PROGRAM Axis03_Y_1
VAR
	Axis03: AXIS_REF;											//회전축
	Axis03_MC_Home: FB_HomeBeforeMoveAX8000;
	Axis03_MC_Power: MC_Power;
	Axis03_Status: MC_ReadStatus;
	Axis03_Position_Read: MC_ReadActualPosition;
	Axis03_Velocity_Read: MC_ReadActualVelocity;
	Axis03_Reset: MC_Reset;										//모터 알람 리셋
	Axis03_Stop: MC_Stop;										//모터 정지
	Axis03_Press_Move: MC_MoveAbsolute;
	Axis03_Home_Pos_Move: MC_MoveAbsolute;
	Axis03_Wait_Pos_Move: MC_MoveAbsolute;
	Axis03_Target_Pos_Move: MC_MoveAbsolute;
	Axis03_Work_End_Move: MC_MoveAbsolute;
	Axis03_Jog: MC_Jog;	
	
	
	Always_ON	:	BOOL	:=TRUE	;//상시 ON
	Always_OFF	:	BOOL	:=FALSE	;//상시 OFF
	Home_Interlock			:	BOOL	;
	Home_Pos_Interlock		: 	BOOL	;
	Wait_Pos_Interlock		:	BOOL	;
	Target_Pos_Interlock	:	BOOL	;
	Work_End_POs_Interlock	:	BOOL	;

	Axis03_Calibration: MC_MoveAbsolute;
	Axis03_Tool_Change: MC_MoveAbsolute;
END_VAR
VAR // added by the converter: edge detectors and wires of the graphical bodies
    _rt1, _rt2, _rt3, _rt4, _rt5 : R_TRIG;
    _w1, _w2 : BOOL;
END_VAR

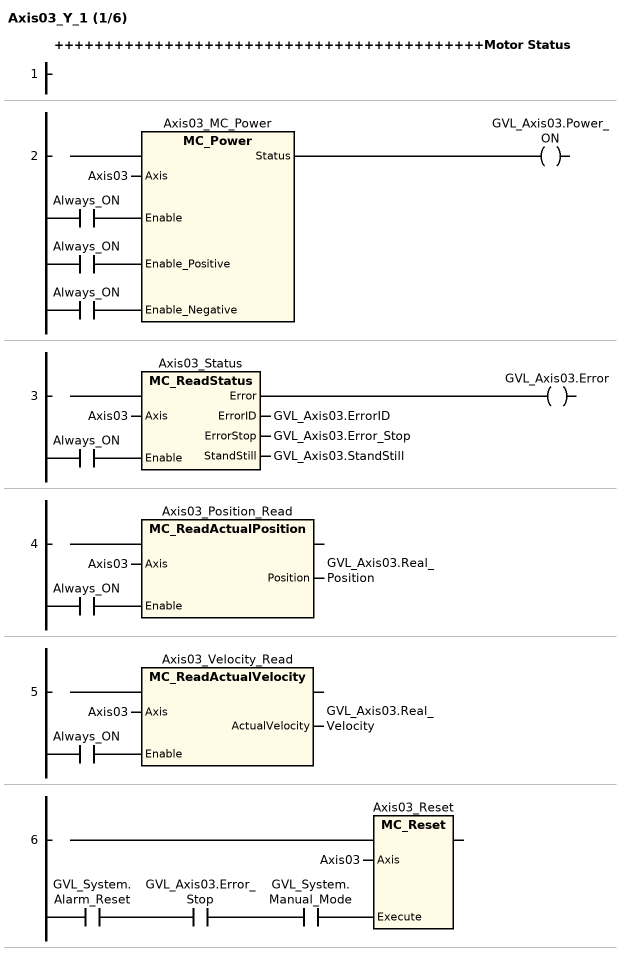
// NETWORK 1: +++++++++++++++++++++++++++++++++++++++++++Motor Status

// NETWORK 2
Axis03_MC_Power(
    Axis := Axis03,
    Enable := Always_ON,
    Enable_Positive := Always_ON,
    Enable_Negative := Always_ON); // MC_Power
GVL_Axis03.Power_ON := Axis03_MC_Power.Status;

// NETWORK 3
Axis03_Status(
    Axis := Axis03,
    Enable := Always_ON,
    Error => GVL_Axis03.Error,
    ErrorID => GVL_Axis03.ErrorID,
    ErrorStop => GVL_Axis03.Error_Stop,
    StandStill => GVL_Axis03.StandStill); // MC_ReadStatus

// NETWORK 4
Axis03_Position_Read(Axis := Axis03, Enable := Always_ON, Position => GVL_Axis03.Real_Position); // MC_ReadActualPosition

// NETWORK 5
Axis03_Velocity_Read(Axis := Axis03, Enable := Always_ON, ActualVelocity => GVL_Axis03.Real_Velocity); // MC_ReadActualVelocity

// NETWORK 6
Axis03_Reset(Axis := Axis03, Execute := GVL_System.Alarm_Reset AND GVL_Axis03.Error_Stop AND GVL_System.Manual_Mode); // MC_Reset

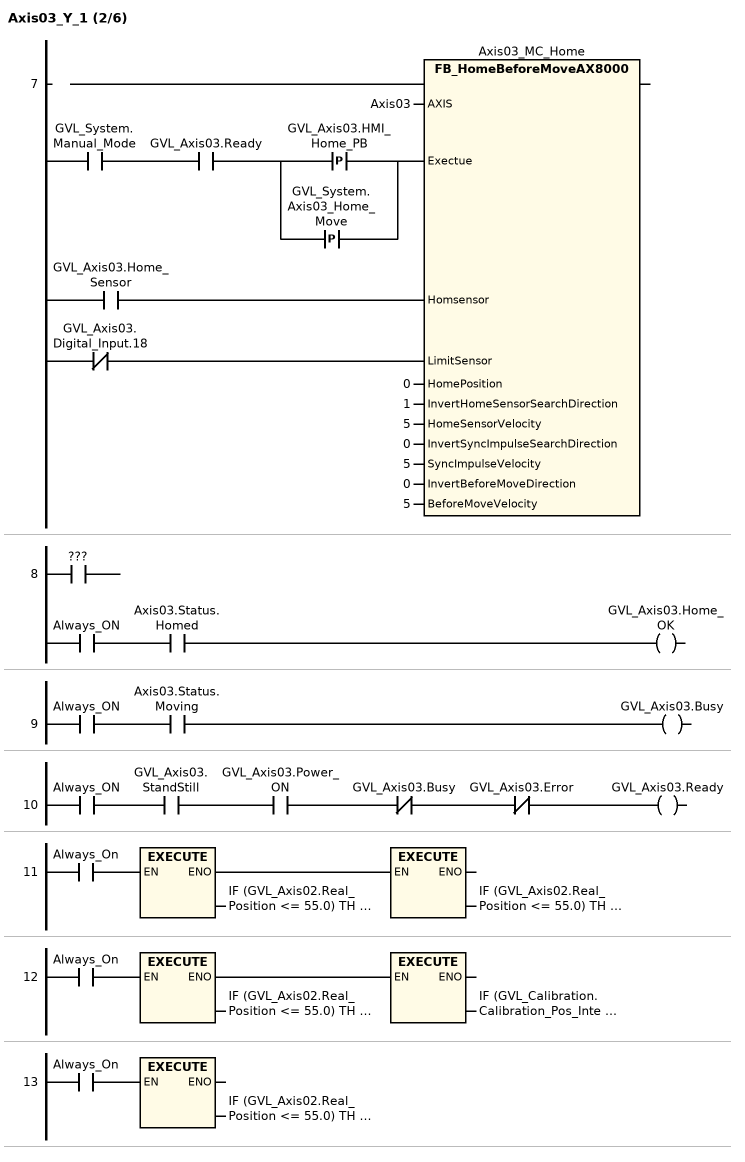
// NETWORK 7
_rt1(CLK := GVL_Axis03.HMI_Home_PB);
_rt2(CLK := GVL_System.Axis03_Home_Move);
Axis03_MC_Home(
    AXIS := Axis03,
    Exectue := GVL_System.Manual_Mode AND GVL_Axis03.Ready AND (_rt1.Q OR _rt2.Q),
    Homsensor := GVL_Axis03.Home_Sensor,
    LimitSensor := NOT GVL_Axis03.Digital_Input.18,
    HomePosition := 0,
    InvertHomeSensorSearchDirection := 1,
    HomeSensorVelocity := 5,
    InvertSyncImpulseSearchDirection := 0,
    SyncImpulseVelocity := 5,
    InvertBeforeMoveDirection := 0,
    BeforeMoveVelocity := 5); // FB_HomeBeforeMoveAX8000

// NETWORK 8
GVL_Axis03.Home_OK := Always_ON AND Axis03.Status.Homed;

// NETWORK 9
GVL_Axis03.Busy := Always_ON AND Axis03.Status.Moving;

// NETWORK 10
GVL_Axis03.Ready := Always_ON AND GVL_Axis03.StandStill AND GVL_Axis03.Power_ON AND NOT GVL_Axis03.Busy AND NOT GVL_Axis03.Error;

// NETWORK 11
_w1 := Always_On;
IF _w1 THEN
    IF (GVL_Axis02.Real_Position <= 55.0) THEN
        Home_Pos_Interlock := TRUE;
    ELSE
        IF (GVL_Axis03.Home_Position_Data >= 12.1) AND 
           (GVL_Axis03.Home_Position_Data <= 18.1) THEN
            Home_Pos_Interlock := TRUE;
        ELSE 
           Home_Pos_Interlock := FALSE;
        END_IF;
    END_IF;
END_IF
IF _w1 THEN
    IF (GVL_Axis02.Real_Position <= 55.0) THEN
        Wait_Pos_Interlock := TRUE;
    ELSE
        IF (GVL_Axis03.Wait_Position_Data >= 12.1) AND 
           (GVL_Axis03.Wait_Position_Data <= 18.1) THEN
            Wait_Pos_Interlock := TRUE;
        ELSE 
           Wait_Pos_Interlock := FALSE;
        END_IF;
    END_IF;
END_IF

// NETWORK 12
_w2 := Always_On;
IF _w2 THEN
    IF (GVL_Axis02.Real_Position <= 55.0) THEN
        Work_End_Pos_Interlock := TRUE;
    ELSE
        IF (GVL_Axis03.Work_End_Position_Data >= 12.1) AND 
           (GVL_Axis03.Work_End_Position_Data <= 18.1) THEN
            Work_End_Pos_Interlock := TRUE;
        ELSE 
           Work_End_Pos_Interlock := FALSE;
        END_IF;
    END_IF;
END_IF
IF _w2 THEN
    IF (GVL_Calibration.Calibration_Pos_Interlock = TRUE) AND (Home_Pos_Interlock = TRUE)
    AND (Wait_Pos_Interlock = TRUE) AND (Target_Pos_Interlock = TRUE) AND (Work_End_POs_Interlock = TRUE) THEN
    	GVL_Axis03.Interlock := TRUE;
    	ELSE
    	GVL_Axis03.Interlock := FALSE;	
    
    END_IF
END_IF

// NETWORK 13
IF Always_On THEN
    IF (GVL_Axis02.Real_Position <= 55.0) THEN
        Home_Interlock := TRUE;
    ELSE
        Home_Interlock := FALSE;
    
    END_IF;
END_IF

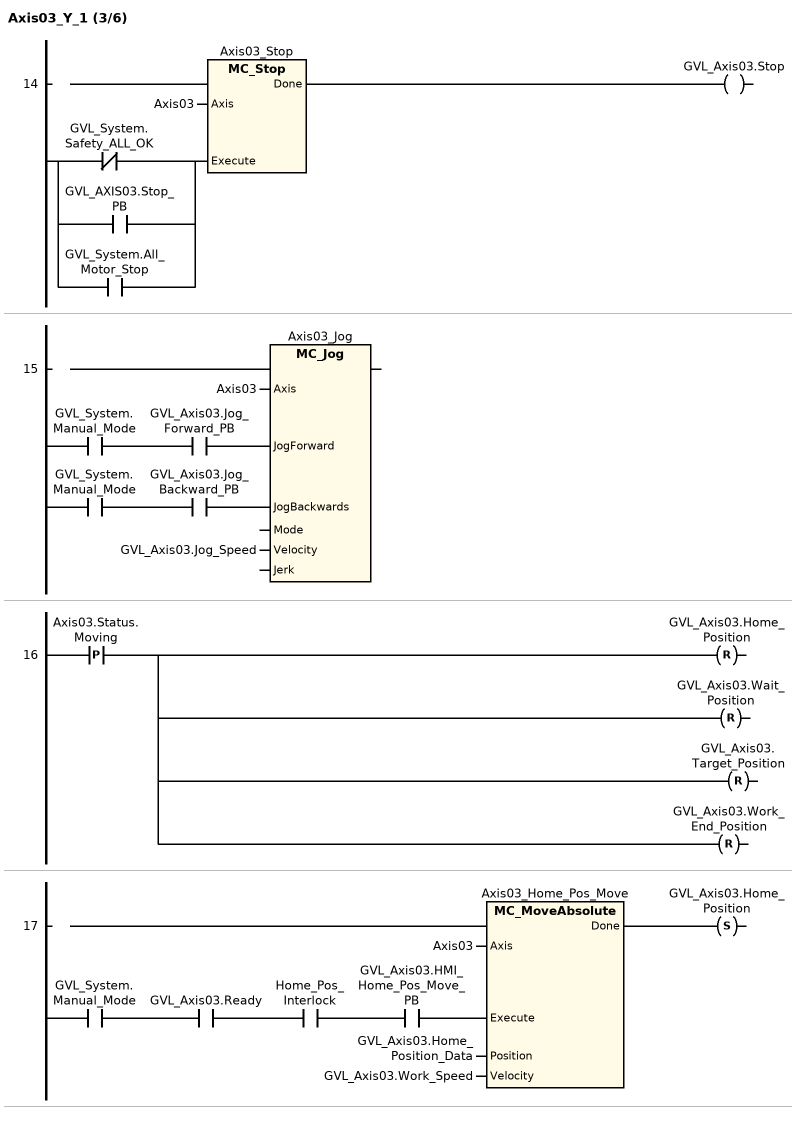
// NETWORK 14
Axis03_Stop(Axis := Axis03, Execute := NOT GVL_System.Safety_ALL_OK OR GVL_AXIS03.Stop_PB OR GVL_System.All_Motor_Stop); // MC_Stop
GVL_Axis03.Stop := Axis03_Stop.Done;

// NETWORK 15
Axis03_Jog(
    Axis := Axis03,
    JogForward := GVL_System.Manual_Mode AND GVL_Axis03.Jog_Forward_PB,
    JogBackwards := GVL_System.Manual_Mode AND GVL_Axis03.Jog_Backward_PB,
    Velocity := GVL_Axis03.Jog_Speed); // MC_Jog

// NETWORK 16
_rt3(CLK := Axis03.Status.Moving);
GVL_Axis03.Home_Position R= _rt3.Q;
GVL_Axis03.Wait_Position R= _rt3.Q;
GVL_Axis03.Target_Position R= _rt3.Q;
GVL_Axis03.Work_End_Position R= _rt3.Q;

// NETWORK 17
Axis03_Home_Pos_Move(
    Axis := Axis03,
    Execute := GVL_System.Manual_Mode AND GVL_Axis03.Ready AND Home_Pos_Interlock AND GVL_Axis03.HMI_Home_Pos_Move_PB,
    Position := GVL_Axis03.Home_Position_Data,
    Velocity := GVL_Axis03.Work_Speed); // MC_MoveAbsolute
GVL_Axis03.Home_Position S= Axis03_Home_Pos_Move.Done;

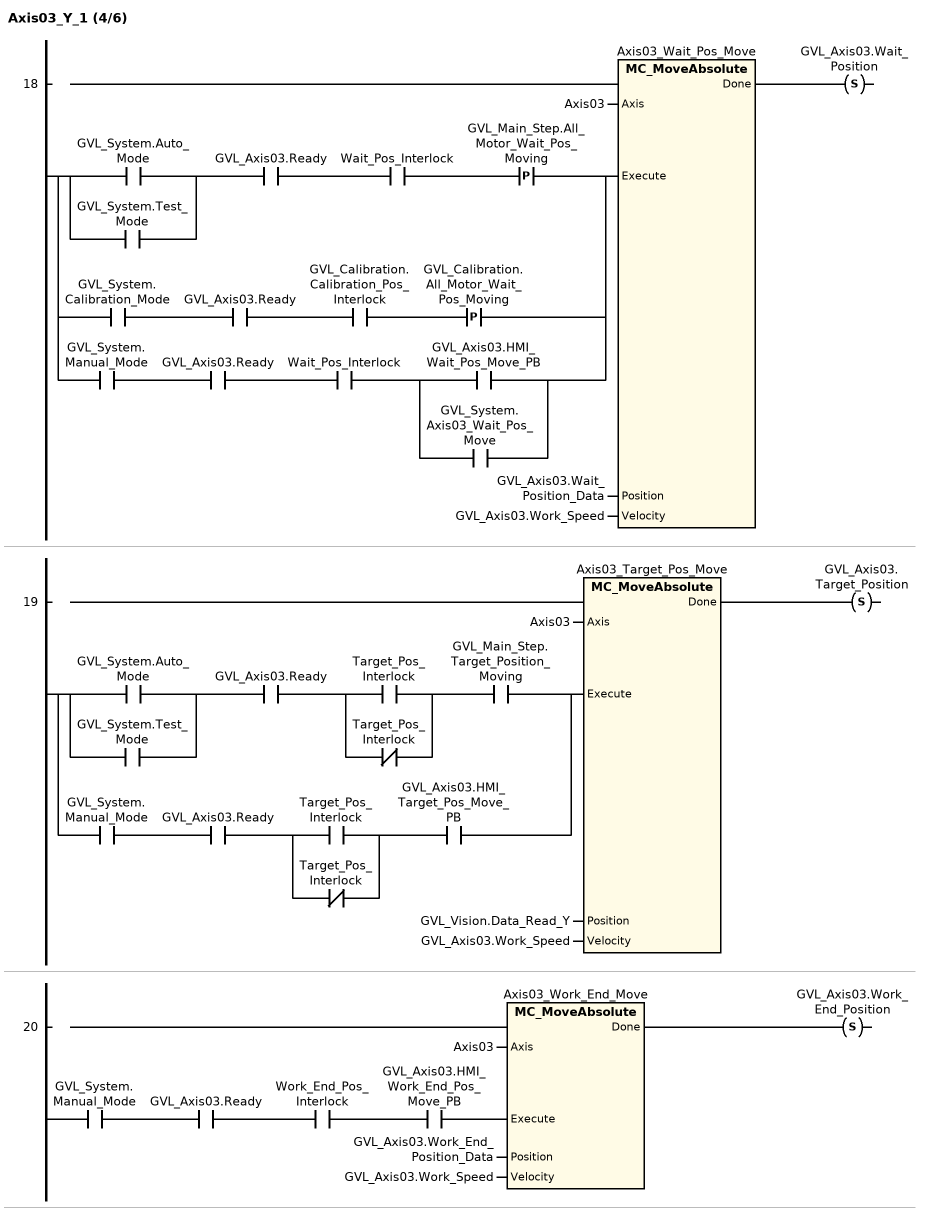
// NETWORK 18
_rt4(CLK := GVL_Main_Step.All_Motor_Wait_Pos_Moving);
_rt5(CLK := GVL_Calibration.All_Motor_Wait_Pos_Moving);
Axis03_Wait_Pos_Move(
    Axis := Axis03,
    Execute := (GVL_System.Auto_Mode OR GVL_System.Test_Mode) AND GVL_Axis03.Ready AND Wait_Pos_Interlock AND _rt4.Q OR GVL_System.Calibration_Mode AND GVL_Axis03.Ready AND GVL_Calibration.Calibration_Pos_Interlock AND _rt5.Q OR GVL_System.Manual_Mode AND GVL_Axis03.Ready AND Wait_Pos_Interlock AND (GVL_Axis03.HMI_Wait_Pos_Move_PB OR GVL_System.Axis03_Wait_Pos_Move),
    Position := GVL_Axis03.Wait_Position_Data,
    Velocity := GVL_Axis03.Work_Speed); // MC_MoveAbsolute
GVL_Axis03.Wait_Position S= Axis03_Wait_Pos_Move.Done;

// NETWORK 19
Axis03_Target_Pos_Move(
    Axis := Axis03,
    Execute := (GVL_System.Auto_Mode OR GVL_System.Test_Mode) AND GVL_Axis03.Ready AND (Target_Pos_Interlock OR NOT Target_Pos_Interlock) AND GVL_Main_Step.Target_Position_Moving OR GVL_System.Manual_Mode AND GVL_Axis03.Ready AND (Target_Pos_Interlock OR NOT Target_Pos_Interlock) AND GVL_Axis03.HMI_Target_Pos_Move_PB,
    Position := GVL_Vision.Data_Read_Y,
    Velocity := GVL_Axis03.Work_Speed); // MC_MoveAbsolute
GVL_Axis03.Target_Position S= Axis03_Target_Pos_Move.Done;

// NETWORK 20
Axis03_Work_End_Move(
    Axis := Axis03,
    Execute := GVL_System.Manual_Mode AND GVL_Axis03.Ready AND Work_End_Pos_Interlock AND GVL_Axis03.HMI_Work_End_Pos_Move_PB,
    Position := GVL_Axis03.Work_End_Position_Data,
    Velocity := GVL_Axis03.Work_Speed); // MC_MoveAbsolute
GVL_Axis03.Work_End_Position S= Axis03_Work_End_Move.Done;

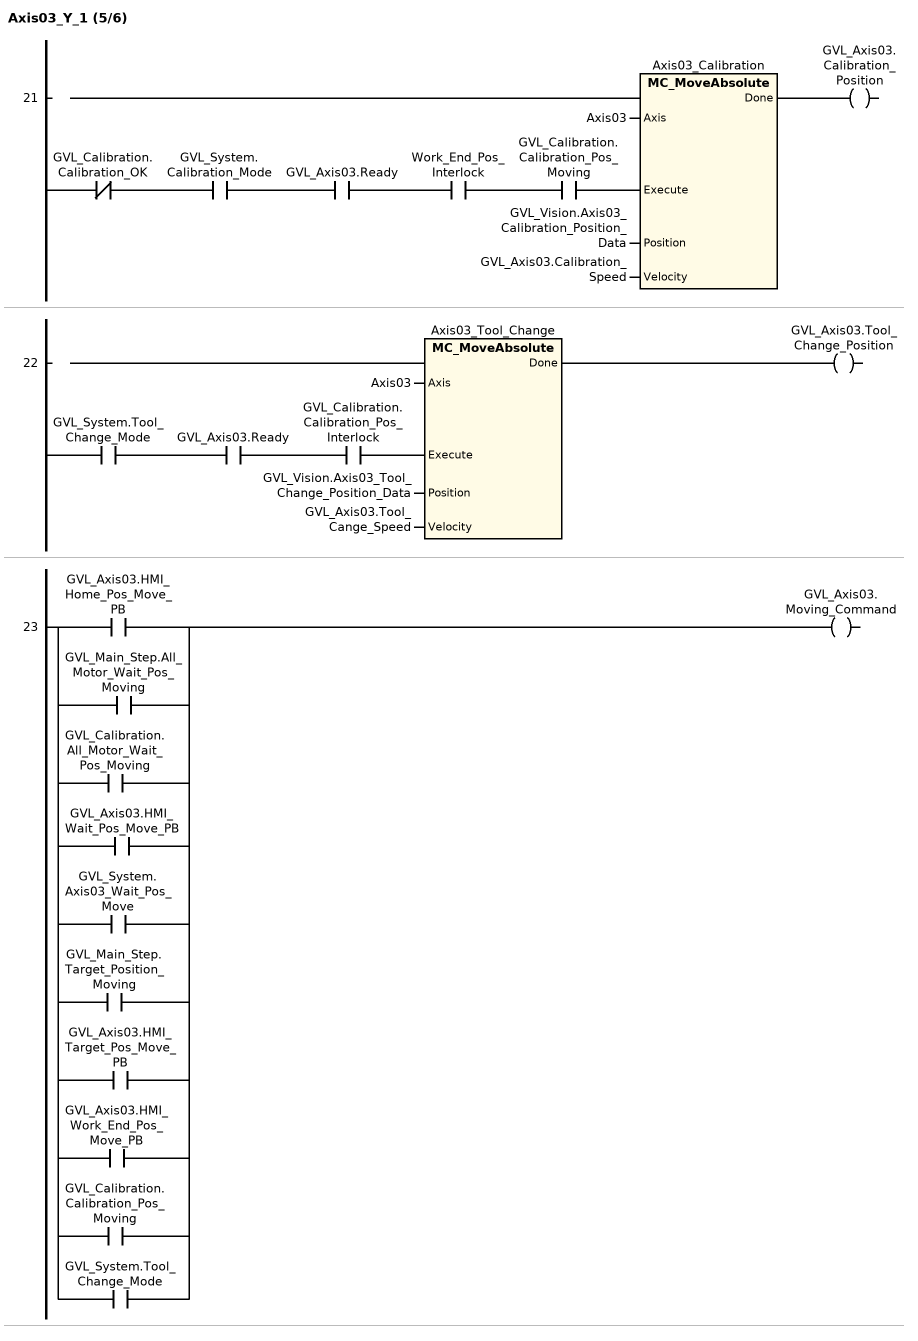
// NETWORK 21
Axis03_Calibration(
    Axis := Axis03,
    Execute := NOT GVL_Calibration.Calibration_OK AND GVL_System.Calibration_Mode AND GVL_Axis03.Ready AND Work_End_Pos_Interlock AND GVL_Calibration.Calibration_Pos_Moving,
    Position := GVL_Vision.Axis03_Calibration_Position_Data,
    Velocity := GVL_Axis03.Calibration_Speed); // MC_MoveAbsolute
GVL_Axis03.Calibration_Position := Axis03_Calibration.Done;

// NETWORK 22
Axis03_Tool_Change(
    Axis := Axis03,
    Execute := GVL_System.Tool_Change_Mode AND GVL_Axis03.Ready AND GVL_Calibration.Calibration_Pos_Interlock,
    Position := GVL_Vision.Axis03_Tool_Change_Position_Data,
    Velocity := GVL_Axis03.Tool_Cange_Speed); // MC_MoveAbsolute
GVL_Axis03.Tool_Change_Position := Axis03_Tool_Change.Done;

// NETWORK 23
GVL_Axis03.Moving_Command := GVL_Axis03.HMI_Home_Pos_Move_PB OR GVL_Main_Step.All_Motor_Wait_Pos_Moving OR GVL_Calibration.All_Motor_Wait_Pos_Moving OR GVL_Axis03.HMI_Wait_Pos_Move_PB OR GVL_System.Axis03_Wait_Pos_Move OR GVL_Main_Step.Target_Position_Moving OR GVL_Axis03.HMI_Target_Pos_Move_PB OR GVL_Axis03.HMI_Work_End_Pos_Move_PB OR GVL_Calibration.Calibration_Pos_Moving OR GVL_System.Tool_Change_Mode;

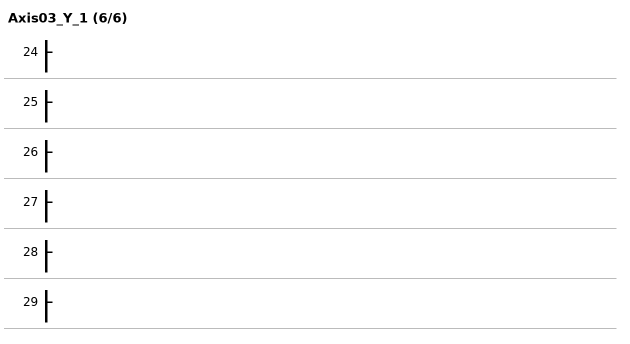
// NETWORK 24

// NETWORK 25

// NETWORK 26

// NETWORK 27

// NETWORK 28

// NETWORK 29

END_PROGRAM

(* stored: Version 1.1.0.1, ProductVersion 3.1.4024.15
   POU Axis03_Y_1: Id {9b7b9669-28f9-40e2-8afc-1b77092ea3a5}, SpecialFunc None *)
